# EPICS autosave request: iocBoot/ioc13Win32/auto_settings.req
file "ccd_settings.req",                P=13Win32:, C=ccd1
file "scan_settings.req",               P=13Win32:, S=scan1
file "scan_settings.req",               P=13Win32:, S=scan2
file "scan_settings.req",               P=13Win32:, S=scan3
file "scan_settings.req",               P=13Win32:, S=scan4
file "CARS_motor_settings.req",         P=13Win32:, M=m1
file "CARS_motor_settings.req",         P=13Win32:, M=m2
file "CARS_motor_settings.req",         P=13Win32:, M=m3
